(* CODESYS project Ladder_and_ST.project

Project tree, tasks and I/O mapping:
  Device : CODESYS Control Win V3, 3S - Smart Software Solutions GmbH, order no. 305021, version 3.5.10.30
    application Application
      libraries: Standard, * (System)
      task MainTask (cyclic, interval t#20ms, priority 1) calls PLC_PRG, PLC2_POU
      task VISU_TASK (cyclic, interval 100 ms, priority 31) calls VisuElems.Visu_Prg
      program PLC_PRG [LD]
      visualisation Visualization
      program PLC2_POU [ST]
  text list GlobalTextList
*)

// Device/Application/PLC_PRG
PROGRAM PLC_PRG
VAR
	Contact1: BOOL;
	Coil1: BOOL;
END_VAR

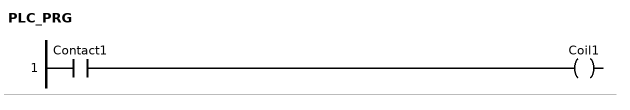
// NETWORK 1
Coil1 := Contact1;

END_PROGRAM

// Device/Application/PLC2_POU
PROGRAM PLC2_POU
VAR
	Contact2: BOOL;
	Coil2: BOOL;
END_VAR

IF Contact2 = TRUE THEN
	Coil2 := TRUE;
ELSE
	Coil2 := FALSE;
END_IF

END_PROGRAM

// Device/Application/Visualization
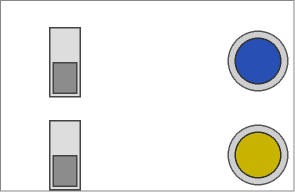
VISUALIZATION Visualization  // 295x192
    DipSwitch (30,27 70x70), variable: PLC_PRG.Contact1, behaviour: TOGGLE, style: Switch-DipSwitch-Gray
    Lamp1 (223,26 70x70), variable: PLC_PRG.Coil1, style: Lamp-Lamp1-Blue
    Lamp1 (223,120 70x70), variable: PLC2_POU.Coil2, style: Lamp-Lamp1-Yellow
    DipSwitch (30,120 70x70), variable: PLC2_POU.Contact2, behaviour: TOGGLE, style: Switch-DipSwitch-Gray
END_VISUALIZATION
